TYPE DUT_IO_Valve01 :
STRUCT
	I_isOpen AT %I* : BOOL := FALSE;
	I_isClosed AT %I*   : BOOL := FALSE;
	I_isHealthy AT %I* : BOOL := FALSE;
	O_setOpen AT %Q*   : BOOL := FALSE;
END_STRUCT
END_TYPE

(* stored: Version 1.1.0.1, ProductVersion 3.1.4024.12
   DUT DUT_IO_Valve01: Id {bcab29c5-b057-4a7d-8b92-5d4128defdf4} *)
